PROGRAM p_AutoWash
VAR

	

END_VAR

END_PROGRAM

(* stored: Version 1.1.0.1, ProductVersion 3.1.4022.18
   POU p_AutoWash: Id {eeb4ee5f-aab1-4444-bdaf-78e7ac6c9f3d}, SpecialFunc None *)
